// TIA Portal V20 export
FUNCTION_BLOCK "Type_6"   // FB7, GRAPH
// stored: GraphVersion 2.0, SetENOAutomatically false
   // inherited from GRAPH_BASE
   VAR_INPUT
      OFF_SQ { ExternalAccessible := 'False'; ExternalVisible := 'False'; ExternalWritable := 'False'} : Bool := false;   // Turn sequence off
      INIT_SQ { ExternalAccessible := 'False'; ExternalVisible := 'False'; ExternalWritable := 'False'} : Bool := false;   // Set sequence to initial state
      ACK_EF { ExternalAccessible := 'False'; ExternalVisible := 'False'; ExternalWritable := 'False'} : Bool := false;   // Acknowledge all errors and faults
      S_PREV { ExternalAccessible := 'False'; ExternalVisible := 'False'; ExternalWritable := 'False'} : Bool := false;   // Output previous step in parameter S_NO
      S_NEXT { ExternalAccessible := 'False'; ExternalVisible := 'False'; ExternalWritable := 'False'} : Bool := false;   // Indicate next step in parameter S_NO
      SW_AUTO { ExternalAccessible := 'False'; ExternalVisible := 'False'; ExternalWritable := 'False'} : Bool := false;   // Automatic mode
      SW_TAP { ExternalAccessible := 'False'; ExternalVisible := 'False'; ExternalWritable := 'False'} : Bool := false;   // Semiautomatic/switch with transition
      SW_TOP { ExternalAccessible := 'False'; ExternalVisible := 'False'; ExternalWritable := 'False'} : Bool := false;   // Semiautomatic/ignore transition
      SW_MAN { ExternalAccessible := 'False'; ExternalVisible := 'False'; ExternalWritable := 'False'} : Bool := false;   // Manual mode
      S_SEL { ExternalAccessible := 'False'; ExternalVisible := 'False'; ExternalWritable := 'False'} : Int := 0;   // Select step to be output to S_NO
      S_ON { ExternalAccessible := 'False'; ExternalVisible := 'False'; ExternalWritable := 'False'} : Bool := false;   // Activate step indicated in S_NO
      S_OFF { ExternalAccessible := 'False'; ExternalVisible := 'False'; ExternalWritable := 'False'} : Bool := false;   // Disable step indicated in S_NO
      T_PUSH { ExternalAccessible := 'False'; ExternalVisible := 'False'; ExternalWritable := 'False'} : Bool := false;   // Enable transition to switch in semi automatic mode
   END_VAR
   VAR_OUTPUT
      S_NO { ExternalAccessible := 'False'; ExternalVisible := 'False'; ExternalWritable := 'False'} : Int := 0;   // Step number
      S_MORE { ExternalAccessible := 'False'; ExternalVisible := 'False'; ExternalWritable := 'False'} : Bool := false;   // More steps are available and can be shown in S_NO
      S_ACTIVE { ExternalAccessible := 'False'; ExternalVisible := 'False'; ExternalWritable := 'False'} : Bool := false;   // Step indicated in S_NO is active
      ERR_FLT { ExternalAccessible := 'False'; ExternalVisible := 'False'; ExternalWritable := 'False'} : Bool := false;   // Interlock or supervision group error
      AUTO_ON { ExternalAccessible := 'False'; ExternalVisible := 'False'; ExternalWritable := 'False'} : Bool := false;   // Automatic mode is active
      TAP_ON { ExternalAccessible := 'False'; ExternalVisible := 'False'; ExternalWritable := 'False'} : Bool := false;   // Semiautomatic mode/step with transition enabled
      TOP_ON { ExternalAccessible := 'False'; ExternalVisible := 'False'; ExternalWritable := 'False'} : Bool := false;   // Semiautomatic mode/ignore transition enabled
      MAN_ON { ExternalAccessible := 'False'; ExternalVisible := 'False'; ExternalWritable := 'False'} : Bool := false;   // Manual mode is active
   END_VAR
BEGIN
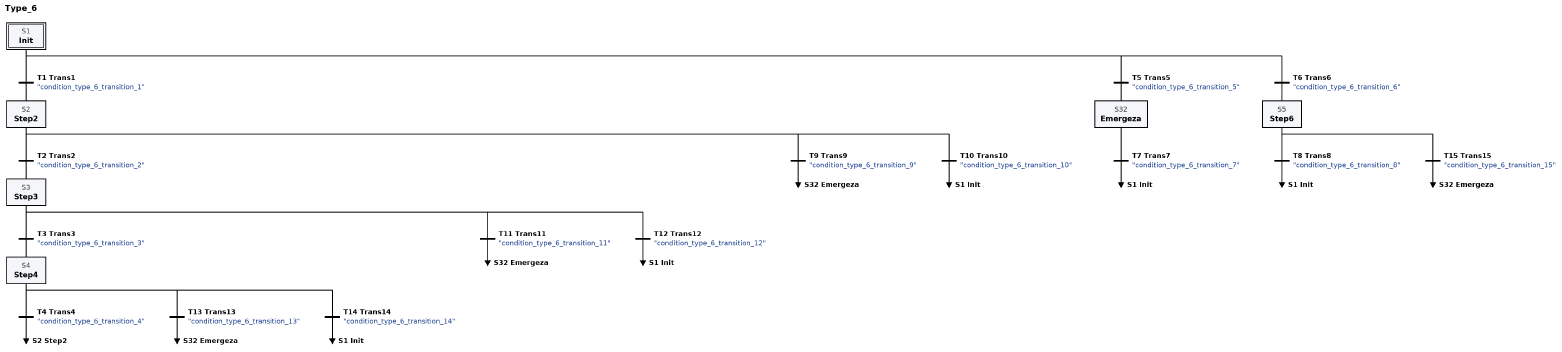
   // sequencer 1
   INITIAL_STEP Init:   // S1, max time T#10S, warning time T#7S
   END_STEP
   TRANSITION Trans1 FROM Init TO Step2   // T1
      := "condition_type_6_transition_1";
   END_TRANSITION
   TRANSITION Trans5 FROM Init TO Emergeza   // T5
      := "condition_type_6_transition_5";
   END_TRANSITION
   TRANSITION Trans6 FROM Init TO Step6   // T6
      := "condition_type_6_transition_6";
   END_TRANSITION
   STEP Step2:   // S2, max time T#10S, warning time T#7S
   END_STEP
   TRANSITION Trans2 FROM Step2 TO Step3   // T2
      := "condition_type_6_transition_2";
   END_TRANSITION
   TRANSITION Trans9 FROM Step2 TO Emergeza   // T9, jump
      := "condition_type_6_transition_9";
   END_TRANSITION
   TRANSITION Trans10 FROM Step2 TO Init   // T10, jump
      := "condition_type_6_transition_10";
   END_TRANSITION
   STEP Step3:   // S3, max time T#10S, warning time T#7S
   END_STEP
   TRANSITION Trans3 FROM Step3 TO Step4   // T3
      := "condition_type_6_transition_3";
   END_TRANSITION
   TRANSITION Trans11 FROM Step3 TO Emergeza   // T11, jump
      := "condition_type_6_transition_11";
   END_TRANSITION
   TRANSITION Trans12 FROM Step3 TO Init   // T12, jump
      := "condition_type_6_transition_12";
   END_TRANSITION
   STEP Step4:   // S4, max time T#10S, warning time T#7S
   END_STEP
   TRANSITION Trans4 FROM Step4 TO Step2   // T4, jump
      := "condition_type_6_transition_4";
   END_TRANSITION
   TRANSITION Trans13 FROM Step4 TO Emergeza   // T13, jump
      := "condition_type_6_transition_13";
   END_TRANSITION
   TRANSITION Trans14 FROM Step4 TO Init   // T14, jump
      := "condition_type_6_transition_14";
   END_TRANSITION
   STEP Emergeza:   // S32, max time T#10S, warning time T#7S
   END_STEP
   TRANSITION Trans7 FROM Emergeza TO Init   // T7, jump
      := "condition_type_6_transition_7";
   END_TRANSITION
   STEP Step6:   // S5, max time T#10S, warning time T#7S
   END_STEP
   TRANSITION Trans8 FROM Step6 TO Init   // T8, jump
      := "condition_type_6_transition_8";
   END_TRANSITION
   TRANSITION Trans15 FROM Step6 TO Emergeza   // T15, jump
      := "condition_type_6_transition_15";
   END_TRANSITION
END_FUNCTION_BLOCK
